// TIA Portal V18 program export: 0 tag tables, 0 data types, 1 data blocks, 2 code blocks (in call order from the OBs), 0 instance data blocks

DATA_BLOCK "Test_DB"   // DB1
{ S7_Optimized_Access := 'TRUE' }
// stored: MemoryReserve 100
   VAR
      "counter" : UDInt;   // Dilly dally
      test : Bool;
   END_VAR
BEGIN
END_DATA_BLOCK

ORGANIZATION_BLOCK "Main"   // OB1, LAD, ProgramCycle
TITLE = "Main Program Sweep (Cycle)"
{ S7_Optimized_Access := 'TRUE' }
// stored: SetENOAutomatically false
   VAR_INPUT
      Initial_Call : Bool;   // Initial call of this OB
      Remanence : Bool;   // =True, if remanent data are available
   END_VAR
BEGIN

REGION Network 1: Test comment
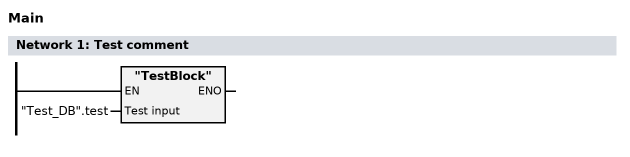
   RUNG wire#powerrail
      "TestBlock"("Test input" := "Test_DB".test)
   END_RUNG
   // the same network as SCL:
   "TestBlock"("Test input" := "Test_DB".test);
END_REGION
END_ORGANIZATION_BLOCK

FUNCTION "TestBlock" : Void   // FC1, LAD
TITLE = What about this?
{ S7_Optimized_Access := 'TRUE' }
// stored: SetENOAutomatically false
   VAR_INPUT
      "Test input" : Bool;   // Hey!
   END_VAR
BEGIN

REGION Network 1: Other test comment
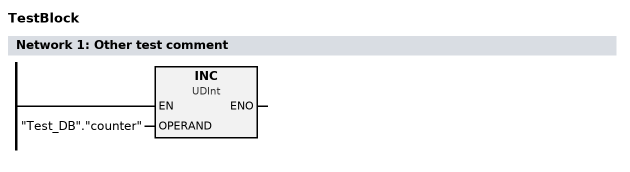
   RUNG wire#powerrail
      { S7_Templates := "DestType := UDInt" } Inc( "Test_DB"."counter" )
   END_RUNG
   // the same network as SCL:
   "Test_DB"."counter" := "Test_DB"."counter" + 1;
END_REGION
END_FUNCTION
